(* PLC project Tc2_IoFunctions.F_SplitDpv1ReadResPkgPNET Demo, tc3-libraries-kb TwinCAT 3.1 *)
(* stored: creationDateTime 2026-05-21T00:00:00, modificationDateTime 2026-05-21T00:00:00 *)

PROGRAM P_Demo_F_SplitDpv1ReadResPkgPNET
  VAR
    aDpv1ReadResBuffer : ARRAY[1..240] OF BYTE;  (* 响应缓冲 *)
    arrDpv1ReqParams : ARRAY[1..39] OF ST_Dpv1ParamAddrEx;  (* 请求清单 *)
    arrDpv1ValueHdr : ARRAY[1..39] OF ST_Dpv1ValueHeaderEx;  (* 解析输出 *)
    bSplitReadResPkgPNET : BOOL := FALSE;  (* 触发解析 *)
    nReadResPkgLenPNET : USINT;  (* 响应长度 *)
  END_VAR

// =============================================================================
// 场景：Profinet SINAMICS 读响应解析。
// 价值：对称封装。
// 验证：收到响应后 bSplitReadResPkgPNET := TRUE → nReadResPkgLenPNET > 0。
// 验证步骤：
//   1. 右键 PLC 项目 → Import PLCopenXML → 选本文件
//   2. 引用 Tc2_IoFunctions（References → Add library）
//   3. 编译 → 登录 → 运行；按上方『验证』行的指示在线写值观察
// =============================================================================

IF bSplitReadResPkgPNET THEN
    nReadResPkgLenPNET := F_SplitDpv1ReadResPkgPNET(
        pDpv1ResData        := ADR(aDpv1ReadResBuffer),
        stDpv1Parameter     := arrDpv1ReqParams,
        stDpv1ValueHeaderEx := arrDpv1ValueHdr
    );
    bSplitReadResPkgPNET := FALSE;
END_IF;
END_PROGRAM
